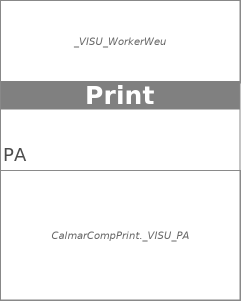
VISUALIZATION _VISU_WorkerWeu_Print  // 241x301
VAR_IN_OUT
  m_Inst : FB_WorkerWeu_Print;
END_VAR
    Frame (0,0 241x83)
        shows _VISU_WorkerWeu(m_Inst := m_Inst)
    Label (0,140 240x30), "PA"
    Rectangle (0,80 240x30), "Print"
    Frame (0,170 241x131)
        shows CalmarCompPrint._VISU_PA(m_Inst := m_Inst.fbPa)
END_VISUALIZATION

(* stored: Version 1.1.0.1, ProductVersion 3.1.4024.11
   Visu _VISU_WorkerWeu_Print: Id {106bf08b-3246-4506-8c48-e81ae7b17b40} *)
